Fanuc KAREL source: kb00034.KL

PROGRAM KB00034
%STACKSIZE=65535
%PRIORITY=65535
%NOLOCKGROUP
VAR
P2 : STRING[80]
-- UNRESOLVED DECLARATIONS (source type spelling not recovered)
-- P1 : TYPE_0x001C (type_u16=0x001C)
BEGIN
P2='A'
CNV_CONF_STR(P1,P2)
END KB00034
